FUNCTION_BLOCK PUBLIC PAEThermistor EXTENDS PAESensorDigital
VAR_INPUT
END_VAR
VAR_OUTPUT
END_VAR
VAR
END_VAR

END_FUNCTION_BLOCK

(* stored: Version 1.1.0.1, ProductVersion 3.1.4020.6
   POU PAEThermistor: Id {92ddab4d-7dd0-48a3-a8a6-57b1a7673cca}, SpecialFunc None *)
